// TIA Portal V19 export
TYPE "FCP_OUT"
   STRUCT
      EFCControlWord { S7_SetPoint := 'True'} : "EFC_CONTROL_WORD";
      FcPControlWord { S7_SetPoint := 'True'} : "FCP_CONTROL_WORD";
      PressureCmd : Word;
      FlowCmd : Word;
   END_STRUCT;
END_TYPE
